INTERFACE IExampleInterface EXTENDS __SYSTEM.IQueryInterface

END_INTERFACE

(* stored: Version 1.1.0.1, ProductVersion 3.1.4024.3
   Itf IExampleInterface: Id {ed62982c-066b-41f3-8c85-24fc99776d86} *)
